# EPICS autosave request: IMMApp/Db/NDPluginSparse_settings.req
file "NDPluginBase_settings.req", P=$(P), R=$(R)
$(P)$(R)Threshold
$(P)$(R)MaxArrayLength
